INTERFACE I_EventHandler_OnExecutionAborted EXTENDS I_EventHandlerBase

METHOD OnExecutionAborted
VAR_INPUT
    Message : T_MaxString;
END_VAR
END_METHOD

END_INTERFACE

(* stored: Version 1.1.0.1, ProductVersion 3.1.4024.4
   Itf I_EventHandler_OnExecutionAborted: Id {b9ba4156-6b91-4bc7-b56d-33c0292aa868}
   Method OnExecutionAborted: Id {85443cfb-8df0-097b-0390-c000c15edbce} *)
